SUBAPPLICATION AuxInput_Seitenschieber_UP (* Subapplication Type *)
  (* Standard: 61499-2 *)
  (* Version 1.0, 2023-02-06, franz *)
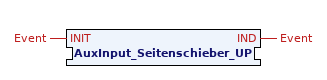
  EVENT_INPUT
    INIT;
  END_EVENT
  EVENT_OUTPUT
    IND;
  END_EVENT
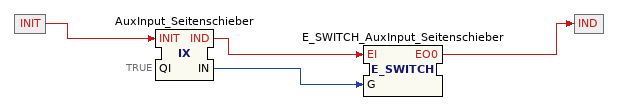
  FBS
    E_SWITCH_AuxInput_Seitenschieber : E_SWITCH;
    AuxInput_Seitenschieber : IX(QI := TRUE);
  END_FBS
  EVENT_CONNECTIONS
    AuxInput_Seitenschieber.IND TO E_SWITCH_AuxInput_Seitenschieber.EI;
    INIT TO AuxInput_Seitenschieber.INIT;
    E_SWITCH_AuxInput_Seitenschieber.EO0 TO IND;
  END_CONNECTIONS
  DATA_CONNECTIONS
    AuxInput_Seitenschieber.IN TO E_SWITCH_AuxInput_Seitenschieber.G;
  END_CONNECTIONS
END_SUBAPPLICATION
